FUNCTION_BLOCK P_Loop (* Runs its body Count times (0 skips it): BODY starts an iteration, NEXT reports its end *)
  (* Standard: 61499-2 *)
  (* Version 2.0, 2026-09-27, Project contributors, Filling cell reference model *)
  PACKAGE fillingcell;
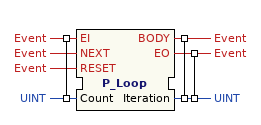
  EVENT_INPUT
    EI WITH Count;
    NEXT;
    RESET;
  END_EVENT
  EVENT_OUTPUT
    BODY WITH Iteration;
    EO WITH Iteration;
  END_EVENT
  VAR_INPUT
    Count : UINT := 1;
  END_VAR
  VAR_OUTPUT
    Iteration : UINT;
  END_VAR
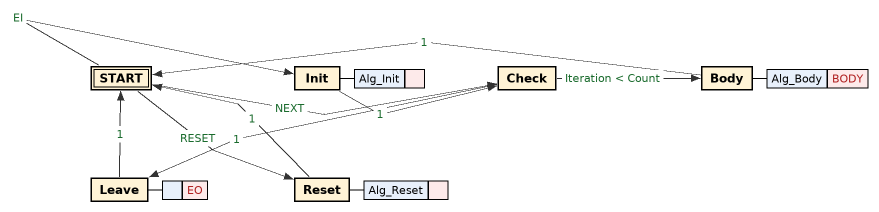
  EC_STATES
    START;
    Init : Alg_Init;
    Check;
    Body : Alg_Body -> BODY;
    Leave : -> EO;
    Reset : Alg_Reset;
  END_STATES
  EC_TRANSITIONS
    START TO Init := EI;
    START TO Check := NEXT;
    START TO Reset := RESET;
    Init TO Check := 1;
    Check TO Body := Iteration < Count;
    Check TO Leave := 1;
    Body TO START := 1;
    Leave TO START := 1;
    Reset TO START := 1;
  END_TRANSITIONS
  ALGORITHM Alg_Init IN ST:
Iteration := 0;
  END_ALGORITHM
  ALGORITHM Alg_Body IN ST:
Iteration := Iteration + 1;
  END_ALGORITHM
  ALGORITHM Alg_Reset IN ST:
Iteration := 0;
  END_ALGORITHM
END_FUNCTION_BLOCK
